Yaskawa INFORM job: A_ROOF_SIDE_0617_1_PL8.JBI

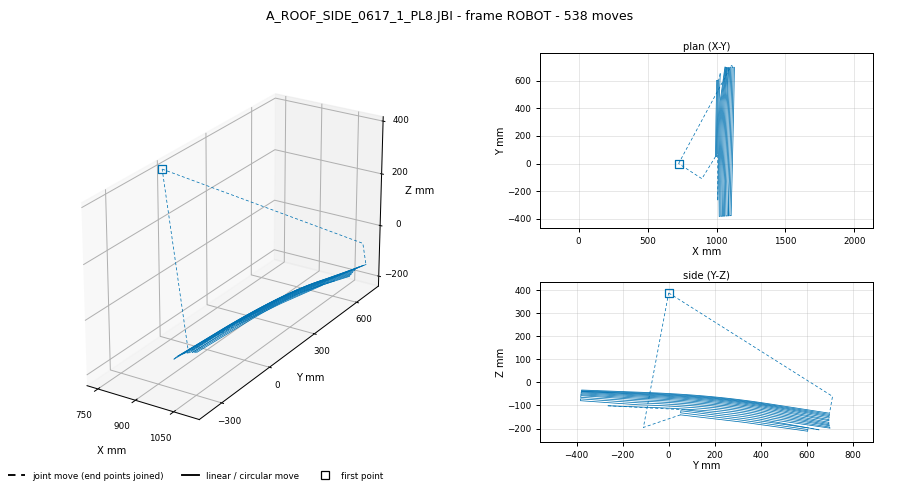
[picture p0: tool path of A_ROOF_SIDE_0617_1_PL8.JBI in frame ROBOT, 538 of 538 moves have a stored position in this frame; points joined in program order, loops and branches not executed]
/JOB
//NAME A_ROOF_SIDE_0617_1_PL8
//POS
///NPOS 538,0,0,0,0,0
///TOOL 0
///USER 0
///POSTYPE ROBOT
///RECTAN
///RCONF 1,0,0,0,0,0,0,0,0,0,0,0,0,0,0,0,0,0,0,0,0,0,0,0
C00000=725.000,0.000,388.500,-180.000,-0.000,0.000
///USER 0
///POSTYPE ROBOT
///RECTAN
C00001=1107.967,711.119,-60.351,170.013,-16.450,1.066
C00002=1129.814,698.090,-133.511,170.013,-16.450,1.066
C00003=1128.918,648.693,-125.824,170.280,-16.606,0.127
C00004=1125.127,440.216,-93.381,170.565,-16.222,-0.283
C00005=1124.690,417.893,-89.964,171.018,-15.554,-0.369
C00006=1124.432,405.287,-88.079,171.255,-15.284,-0.399
C00007=1124.145,391.687,-86.083,171.500,-15.059,-0.421
C00008=1123.832,377.143,-83.997,171.755,-14.880,-0.433
C00009=1123.494,361.710,-81.840,172.018,-14.745,-0.437
C00010=1123.153,346.326,-79.747,172.273,-14.658,-0.434
C00011=1122.809,330.942,-77.713,172.523,-14.609,-0.424
C00012=1122.428,313.994,-75.547,172.790,-14.590,-0.408
C00013=1122.033,296.572,-73.395,173.060,-14.603,-0.387
C00014=1121.637,279.197,-71.328,173.323,-14.640,-0.363
C00015=1121.232,261.424,-69.294,173.585,-14.699,-0.335
C00016=1120.814,243.073,-67.283,173.850,-14.777,-0.305
C00017=1120.393,224.685,-65.353,174.108,-14.866,-0.273
C00018=1119.732,195.801,-62.498,174.517,-15.066,-0.216
C00019=1119.265,175.675,-60.613,174.766,-15.231,-0.174
C00020=1118.801,155.633,-58.834,175.006,-15.376,-0.135
C00021=1118.319,134.585,-57.072,175.249,-15.506,-0.098
C00022=1117.837,113.529,-55.408,175.483,-15.610,-0.064
C00023=1117.332,91.368,-53.767,175.719,-15.694,-0.032
C00024=1116.829,69.300,-52.233,175.943,-15.752,-0.004
C00025=1116.302,46.128,-50.732,176.170,-15.788,0.023
C00026=1115.776,23.049,-49.338,176.385,-15.806,0.048
C00027=1115.222,-1.112,-47.980,176.600,-15.809,0.071
C00028=1114.667,-25.180,-46.725,176.803,-15.805,0.094
C00029=1114.080,-50.322,-45.510,177.003,-15.802,0.117
C00030=1113.487,-75.397,-44.389,177.192,-15.806,0.141
C00031=1112.880,-100.584,-43.344,177.368,-15.827,0.165
C00032=1107.242,-327.548,-34.722,177.586,-15.877,0.062
C00033=1106.000,-377.496,-32.825,177.740,-15.899,-0.498
C00034=1096.541,-377.841,-35.728,177.817,-15.909,-0.779
C00035=1097.765,-327.892,-37.635,177.577,-15.875,0.098
C00036=1103.334,-100.476,-46.316,177.367,-15.826,0.169
C00037=1103.941,-75.303,-47.364,177.191,-15.806,0.144
C00038=1104.536,-50.241,-48.492,177.002,-15.801,0.120
C00039=1105.124,-25.111,-49.715,176.802,-15.805,0.096
C00040=1105.682,-1.059,-50.978,176.599,-15.809,0.073
C00041=1106.238,23.090,-52.343,176.385,-15.805,0.049
C00042=1106.766,46.153,-53.742,176.170,-15.788,0.024
C00043=1107.294,69.311,-55.246,175.943,-15.752,-0.003
C00044=1107.796,91.366,-56.778,175.718,-15.694,-0.032
C00045=1108.299,113.513,-58.415,175.483,-15.610,-0.064
C00046=1108.778,134.556,-60.069,175.249,-15.506,-0.098
C00047=1109.257,155.591,-61.820,175.007,-15.376,-0.136
C00048=1109.716,175.621,-63.583,174.766,-15.231,-0.175
C00049=1110.177,195.736,-65.450,174.517,-15.066,-0.217
C00050=1110.476,208.693,-66.708,174.325,-14.951,-0.246
C00051=1110.835,224.601,-68.294,174.108,-14.866,-0.274
C00052=1111.254,242.975,-70.217,173.850,-14.777,-0.306
C00053=1111.671,261.313,-72.224,173.585,-14.700,-0.337
C00054=1112.076,279.073,-74.255,173.323,-14.641,-0.365
C00055=1112.471,296.435,-76.322,173.061,-14.603,-0.390
C00056=1112.868,313.842,-78.478,172.791,-14.591,-0.411
C00057=1113.252,330.775,-80.653,172.523,-14.609,-0.427
C00058=1113.600,346.143,-82.698,172.274,-14.659,-0.437
C00059=1113.947,361.511,-84.808,172.019,-14.746,-0.441
C00060=1114.293,376.928,-86.991,171.756,-14.880,-0.437
C00061=1114.616,391.453,-89.109,171.501,-15.060,-0.425
C00062=1114.916,405.034,-91.143,171.257,-15.285,-0.405
C00063=1115.190,417.620,-93.073,171.019,-15.554,-0.375
C00064=1115.441,429.264,-94.900,170.787,-15.869,-0.337
C00065=1115.665,439.899,-96.600,170.567,-16.223,-0.290
C00066=1119.956,648.127,-130.473,170.298,-16.616,0.066
C00067=1120.972,697.468,-138.499,169.874,-16.366,1.559
C00068=1112.130,696.831,-143.487,170.053,-16.473,0.925
C00069=1110.996,647.549,-135.122,170.327,-16.632,-0.034
C00070=1106.203,439.581,-99.820,170.569,-16.224,-0.297
C00071=1105.958,428.969,-98.061,170.789,-15.870,-0.343
C00072=1105.690,417.346,-96.183,171.021,-15.555,-0.381
C00073=1105.400,404.781,-94.207,171.258,-15.286,-0.410
C00074=1105.088,391.219,-92.134,171.502,-15.061,-0.430
C00075=1104.754,376.713,-89.984,171.758,-14.881,-0.441
C00076=1104.400,361.312,-87.777,172.020,-14.746,-0.445
C00077=1104.048,345.961,-85.648,172.275,-14.659,-0.440
C00078=1103.695,330.607,-83.592,172.524,-14.610,-0.430
C00079=1103.308,313.689,-81.408,172.791,-14.591,-0.413
C00080=1102.911,296.297,-79.249,173.061,-14.603,-0.392
C00081=1102.515,278.948,-77.182,173.324,-14.641,-0.367
C00082=1102.110,261.203,-75.154,173.586,-14.700,-0.339
C00083=1101.695,242.879,-73.151,173.850,-14.777,-0.308
C00084=1101.278,224.517,-71.234,174.109,-14.867,-0.275
C00085=1100.917,208.619,-69.643,174.325,-14.952,-0.247
C00086=1100.623,195.671,-68.402,174.517,-15.066,-0.218
C00087=1100.167,175.566,-66.553,174.767,-15.231,-0.175
C00088=1099.714,155.549,-64.805,175.007,-15.376,-0.136
C00089=1099.238,134.527,-63.067,175.249,-15.506,-0.098
C00090=1098.762,113.496,-61.421,175.483,-15.610,-0.064
C00091=1098.260,91.363,-59.788,175.718,-15.693,-0.031
C00092=1097.759,69.323,-58.260,175.943,-15.752,-0.002
C00093=1097.230,46.180,-56.752,176.169,-15.788,0.025
C00094=1096.700,23.129,-55.348,176.384,-15.805,0.050
C00095=1096.142,-1.005,-53.975,176.599,-15.809,0.075
C00096=1095.582,-25.044,-52.704,176.802,-15.805,0.098
C00097=1094.991,-50.159,-51.473,177.002,-15.801,0.123
C00098=1094.393,-75.207,-50.339,177.190,-15.806,0.148
C00099=1093.786,-100.367,-49.288,177.366,-15.826,0.173
C00100=1088.286,-328.237,-40.548,177.560,-15.873,0.157
C00101=1087.079,-378.186,-38.632,177.718,-15.896,-0.418
C00102=1088.610,-378.564,-38.329,177.695,-18.663,-0.346
C00103=1087.602,-328.640,-40.895,177.480,-18.637,0.327
C00104=1083.551,-128.437,-51.180,177.438,-18.638,0.450
C00105=1084.148,-103.852,-52.113,177.268,-18.642,0.435
C00106=1084.733,-79.664,-53.112,177.091,-18.674,0.423
C00107=1085.309,-55.600,-54.189,176.905,-18.731,0.414
C00108=1085.881,-31.455,-55.358,176.709,-18.808,0.406
C00109=1086.446,-7.402,-56.613,176.507,-18.895,0.400
C00110=1087.009,16.760,-57.969,176.295,-18.988,0.394
C00111=1087.541,39.825,-59.355,176.086,-19.073,0.389
C00112=1088.069,62.885,-60.834,175.869,-19.149,0.384
C00113=1088.598,86.051,-62.417,175.642,-19.211,0.377
C00114=1089.097,108.100,-64.017,175.419,-19.253,0.369
C00115=1089.596,130.256,-65.721,175.186,-19.276,0.358
C00116=1090.069,151.295,-67.432,174.954,-19.282,0.346
C00117=1090.541,172.325,-69.237,174.713,-19.270,0.332
C00118=1090.993,192.461,-71.058,174.472,-19.248,0.317
C00119=1091.350,208.411,-72.568,174.213,-19.225,0.305
C00120=1091.518,215.896,-73.306,174.110,-19.239,0.302
C00121=1091.934,234.336,-75.185,173.852,-19.278,0.297
C00122=1092.339,252.213,-77.095,173.593,-19.321,0.292
C00123=1092.756,270.561,-79.145,173.319,-19.373,0.289
C00124=1093.151,287.916,-81.174,173.051,-19.435,0.288
C00125=1093.539,304.875,-83.242,172.781,-19.511,0.289
C00126=1093.917,321.322,-85.330,172.510,-19.607,0.295
C00127=1094.297,337.735,-87.498,172.229,-19.729,0.304
C00128=1094.655,353.122,-89.610,171.955,-19.874,0.319
C00129=1094.993,367.519,-91.659,171.687,-20.045,0.338
C00130=1095.333,381.964,-93.787,171.405,-20.259,0.365
C00131=1095.657,395.520,-95.855,171.126,-20.509,0.400
C00132=1095.962,408.134,-97.843,170.850,-20.795,0.441
C00133=1096.246,419.755,-99.732,170.576,-21.115,0.490
C00134=1096.509,430.438,-101.522,170.302,-21.468,0.545
C00135=1096.760,440.397,-103.240,170.025,-21.859,0.609
C00136=1102.067,647.102,-139.894,169.706,-22.284,0.894
C00137=1103.328,696.318,-148.621,169.517,-22.199,1.393
C00138=1095.176,695.746,-154.761,168.937,-27.270,1.833
C00139=1093.722,646.605,-145.650,168.975,-27.285,1.750
C00140=1087.640,441.197,-107.568,169.355,-26.880,1.480
C00141=1087.362,431.351,-105.797,169.700,-26.465,1.400
C00142=1087.070,420.586,-103.925,170.040,-26.078,1.327
C00143=1086.786,409.872,-102.124,170.346,-25.748,1.265
C00144=1086.506,399.019,-100.357,170.629,-25.461,1.212
C00145=1086.184,386.323,-98.356,170.934,-25.175,1.160
C00146=1085.845,372.684,-96.281,171.239,-24.915,1.114
C00147=1085.515,359.148,-94.295,171.522,-24.696,1.075
C00148=1085.166,344.673,-92.247,171.808,-24.495,1.041
C00149=1084.806,329.574,-90.188,172.089,-24.315,1.010
C00150=1084.418,313.062,-88.024,172.381,-24.143,0.982
C00151=1084.033,296.553,-85.949,172.660,-23.990,0.958
C00152=1083.631,279.213,-83.859,172.941,-23.844,0.935
C00153=1083.216,261.139,-81.776,173.221,-23.701,0.914
C00154=1082.793,242.708,-79.747,173.496,-23.562,0.894
C00155=1082.371,224.240,-77.807,173.762,-23.423,0.875
C00156=1082.004,208.130,-76.188,173.986,-23.302,0.859
C00157=1081.621,191.051,-74.571,174.293,-23.234,0.850
C00158=1081.149,170.019,-72.671,174.543,-23.151,0.841
C00159=1080.675,148.977,-70.868,174.780,-23.062,0.831
C00160=1080.175,126.805,-69.067,175.017,-22.959,0.821
C00161=1079.674,104.750,-67.372,175.244,-22.845,0.809
C00162=1079.145,81.692,-65.701,175.472,-22.715,0.796
C00163=1078.611,58.504,-64.117,175.694,-22.574,0.783
C00164=1078.075,35.433,-62.636,175.908,-22.429,0.771
C00165=1077.532,12.237,-61.240,176.119,-22.282,0.759
C00166=1076.988,-10.831,-59.941,176.323,-22.141,0.748
C00167=1076.437,-33.998,-58.724,176.523,-22.011,0.740
C00168=1075.885,-57.066,-57.598,176.719,-21.901,0.734
C00169=1075.327,-80.143,-56.557,176.907,-21.815,0.731
C00170=1074.762,-103.356,-55.591,177.090,-21.760,0.731
C00171=1074.152,-128.448,-54.634,177.278,-21.736,0.736
C00172=1077.280,-329.161,-44.155,177.328,-21.727,0.620
C00173=1078.056,-379.088,-41.549,177.471,-21.743,0.235
C00174=1068.156,-379.602,-45.133,177.168,-25.215,0.859
C00175=1067.520,-329.679,-47.816,177.119,-25.210,0.975
C00176=1064.951,-128.477,-58.631,177.065,-25.228,1.072
C00177=1065.229,-116.921,-59.062,176.973,-25.231,1.075
C00178=1065.772,-94.813,-59.942,176.790,-25.259,1.081
C00179=1066.313,-72.653,-60.902,176.600,-25.321,1.092
C00180=1066.853,-50.507,-61.942,176.405,-25.414,1.106
C00181=1067.390,-28.375,-63.063,176.206,-25.532,1.124
C00182=1067.937,-5.743,-64.294,176.002,-25.673,1.145
C00183=1068.491,17.337,-65.640,175.791,-25.833,1.169
C00184=1069.042,40.486,-67.081,175.577,-26.003,1.196
C00185=1069.589,63.630,-68.614,175.359,-26.177,1.225
C00186=1070.132,86.767,-70.243,175.137,-26.351,1.254
C00187=1070.658,109.399,-71.931,174.912,-26.517,1.284
C00188=1071.167,131.459,-73.669,174.684,-26.676,1.314
C00189=1071.663,153.080,-75.466,174.451,-26.827,1.343
C00190=1072.145,174.194,-77.317,174.211,-26.973,1.373
C00191=1072.611,194.733,-79.211,173.962,-27.116,1.402
C00192=1072.907,207.781,-80.465,173.665,-27.213,1.423
C00193=1073.311,225.064,-82.231,173.424,-27.400,1.459
C00194=1073.745,243.621,-84.215,173.156,-27.596,1.499
C00195=1074.180,262.140,-86.287,172.876,-27.788,1.539
C00196=1074.609,280.284,-88.415,172.589,-27.977,1.580
C00197=1075.028,297.831,-90.565,172.298,-28.165,1.621
C00198=1075.427,314.433,-92.689,172.006,-28.354,1.663
C00199=1075.807,330.049,-94.772,171.717,-28.547,1.706
C00200=1076.185,345.347,-96.894,171.414,-28.755,1.752
C00201=1076.552,359.920,-98.998,171.105,-28.980,1.802
C00202=1076.903,373.558,-101.043,170.793,-29.218,1.856
C00203=1077.239,386.313,-103.027,170.477,-29.476,1.912
C00204=1077.533,397.166,-104.775,170.185,-29.725,1.968
C00205=1077.863,408.975,-106.743,169.837,-30.038,2.037
C00206=1078.176,419.800,-108.614,169.482,-30.369,2.110
C00207=1078.474,429.699,-110.386,169.121,-30.716,2.187
C00208=1078.782,439.524,-112.210,168.717,-31.114,2.275
C00209=1085.876,646.161,-151.960,168.189,-31.575,2.533
C00210=1087.559,695.233,-161.401,168.348,-31.628,2.229
C00211=1085.673,695.022,-166.146,167.623,-35.268,2.859
C00212=1082.684,645.978,-156.885,167.361,-35.185,3.314
C00213=1070.662,448.821,-119.660,167.510,-35.179,3.127
C00214=1070.296,439.181,-117.737,168.020,-34.766,3.021
C00215=1069.983,430.349,-116.040,168.434,-34.434,2.936
C00216=1069.647,420.308,-114.182,168.853,-34.101,2.851
C00217=1069.471,414.833,-113.197,169.061,-33.937,2.808
C00218=1069.131,403.873,-111.284,169.443,-33.640,2.731
C00219=1068.806,392.964,-109.447,169.785,-33.381,2.663
C00220=1068.464,381.099,-107.520,170.122,-33.133,2.597
C00221=1068.095,367.780,-105.438,170.467,-32.888,2.532
C00222=1067.724,354.051,-103.373,170.792,-32.666,2.471
C00223=1067.353,339.856,-101.319,171.102,-32.462,2.414
C00224=1066.964,324.712,-99.214,171.408,-32.264,2.358
C00225=1066.556,308.542,-97.054,171.711,-32.069,2.303
C00226=1066.142,291.850,-94.918,172.005,-31.880,2.250
C00227=1065.720,274.707,-92.814,172.288,-31.692,2.197
C00228=1065.281,256.709,-90.699,172.569,-31.496,2.143
C00229=1064.831,238.191,-88.620,172.845,-31.290,2.088
C00230=1064.475,223.486,-87.033,173.054,-31.121,2.045
C00231=1064.085,207.368,-85.358,173.275,-30.929,1.997
C00232=1063.829,196.371,-84.284,173.586,-30.836,1.971
C00233=1063.364,176.327,-82.401,173.836,-30.678,1.927
C00234=1062.893,156.134,-80.594,174.069,-30.525,1.884
C00235=1062.401,135.075,-78.801,174.300,-30.369,1.841
C00236=1061.880,113.012,-77.019,174.529,-30.207,1.797
C00237=1061.353,90.801,-75.318,174.751,-30.044,1.755
C00238=1060.799,67.727,-73.649,174.975,-29.877,1.712
C00239=1060.262,45.503,-72.130,175.186,-29.719,1.673
C00240=1059.725,23.413,-70.707,175.395,-29.569,1.635
C00241=1059.185,1.324,-69.370,175.602,-29.429,1.600
C00242=1058.639,-20.884,-68.111,175.812,-29.304,1.568
C00243=1058.095,-42.966,-66.946,176.018,-29.200,1.540
C00244=1057.574,-64.054,-65.913,176.216,-29.126,1.516
C00245=1057.052,-85.283,-64.950,176.412,-29.078,1.496
C00246=1056.555,-105.402,-64.111,176.594,-29.061,1.480
C00247=1055.993,-128.515,-63.229,176.797,-29.077,1.467
C00248=1058.090,-330.203,-52.056,176.852,-29.052,1.390
C00249=1058.608,-380.124,-49.292,176.773,-29.044,1.551
C00250=1050.380,-380.614,-53.513,176.302,-33.105,2.273
C00251=1049.775,-330.705,-56.474,176.539,-33.127,1.840
C00252=1047.327,-129.069,-68.445,176.478,-33.153,1.918
C00253=1047.362,-127.070,-68.526,176.459,-33.153,1.920
C00254=1047.879,-105.949,-69.326,176.261,-33.099,1.940
C00255=1048.393,-85.139,-70.194,176.061,-33.077,1.964
C00256=1048.903,-64.584,-71.130,175.861,-33.085,1.991
C00257=1049.429,-43.491,-72.170,175.654,-33.119,2.022
C00258=1049.956,-22.405,-73.293,175.448,-33.176,2.058
C00259=1050.512,-0.188,-74.563,175.233,-33.258,2.098
C00260=1051.064,21.906,-75.914,175.020,-33.355,2.141
C00261=1051.614,43.999,-77.354,174.810,-33.464,2.187
C00262=1052.164,66.232,-78.889,174.597,-33.581,2.235
C00263=1052.706,88.312,-80.504,174.383,-33.703,2.285
C00264=1053.247,110.530,-82.218,174.162,-33.830,2.336
C00265=1053.780,132.597,-84.016,173.934,-33.957,2.388
C00266=1054.285,153.658,-85.822,173.705,-34.082,2.440
C00267=1054.763,173.716,-87.630,173.473,-34.206,2.491
C00268=1055.225,193.096,-89.463,173.230,-34.334,2.542
C00269=1055.554,206.894,-90.825,172.843,-34.435,2.581
C00270=1055.703,212.785,-91.440,172.766,-34.500,2.602
C00271=1056.202,232.613,-93.575,172.496,-34.711,2.671
C00272=1056.671,251.300,-95.681,172.227,-34.899,2.736
C00273=1057.120,269.057,-97.770,171.956,-35.072,2.797
C00274=1057.572,286.820,-99.954,171.667,-35.245,2.860
C00275=1058.004,303.622,-102.108,171.375,-35.412,2.921
C00276=1058.420,319.514,-104.233,171.076,-35.578,2.982
C00277=1058.816,334.373,-106.302,170.775,-35.745,3.042
C00278=1059.221,349.205,-108.450,170.448,-35.929,3.106
C00279=1059.611,363.053,-110.539,170.112,-36.121,3.172
C00280=1059.987,375.974,-112.567,169.769,-36.324,3.238
C00281=1060.351,388.020,-114.531,169.415,-36.538,3.307
C00282=1060.725,399.843,-116.535,169.029,-36.777,3.382
C00283=1061.093,410.950,-118.492,168.625,-37.034,3.461
C00284=1061.448,421.083,-120.350,168.210,-37.301,3.541
C00285=1061.790,430.304,-122.105,167.786,-37.574,3.622
C00286=1062.137,439.125,-123.850,167.329,-37.867,3.709
C00287=1062.510,447.936,-125.662,166.813,-38.196,3.805
C00288=1075.955,645.876,-163.643,166.601,-38.231,3.971
C00289=1079.282,694.871,-173.044,167.101,-38.379,3.164
C00290=1075.415,695.159,-178.337,166.551,-40.986,3.567
C00291=1071.311,646.171,-169.207,165.871,-40.794,4.606
C00292=1054.724,448.260,-132.325,166.101,-40.779,4.434
C00293=1054.610,446.311,-131.924,166.230,-40.722,4.414
C00294=1054.216,437.743,-130.128,166.759,-40.461,4.326
C00295=1053.840,428.947,-128.357,167.239,-40.220,4.244
C00296=1053.448,419.135,-126.460,167.713,-39.981,4.161
C00297=1053.061,408.824,-124.545,168.154,-39.759,4.081
C00298=1052.661,397.544,-122.535,168.582,-39.546,4.003
C00299=1052.286,386.328,-120.613,168.963,-39.360,3.932
C00300=1051.899,374.242,-118.621,169.332,-39.185,3.863
C00301=1051.506,361.410,-116.588,169.686,-39.023,3.795
C00302=1051.093,347.398,-114.456,170.034,-38.867,3.728
C00303=1050.695,333.396,-112.407,170.350,-38.730,3.665
C00304=1050.274,318.188,-110.271,170.663,-38.597,3.601
C00305=1049.840,302.168,-108.112,170.966,-38.470,3.537
C00306=1049.388,285.212,-105.920,171.260,-38.344,3.472
C00307=1048.917,267.295,-103.701,171.545,-38.216,3.406
C00308=1048.448,249.385,-101.576,171.812,-38.088,3.341
C00309=1047.955,230.394,-99.417,172.076,-37.947,3.271
C00310=1047.327,206.362,-96.817,172.388,-37.756,3.183
C00311=1046.886,188.254,-95.024,172.868,-37.679,3.129
C00312=1046.398,168.205,-93.133,173.114,-37.609,3.074
C00313=1045.906,147.976,-91.318,173.343,-37.549,3.021
C00314=1045.370,126.086,-89.451,173.574,-37.490,2.965
C00315=1044.822,103.869,-87.653,173.797,-37.436,2.909
C00316=1044.273,81.793,-85.961,174.011,-37.389,2.856
C00317=1043.717,59.563,-84.348,174.222,-37.345,2.803
C00318=1043.160,37.472,-82.836,174.431,-37.309,2.753
C00319=1042.600,15.376,-81.412,174.641,-37.283,2.704
C00320=1042.062,-5.859,-80.127,174.847,-37.271,2.660
C00321=1041.529,-26.948,-78.935,175.054,-37.274,2.618
C00322=1040.998,-48.038,-77.827,175.265,-37.297,2.579
C00323=1040.491,-68.268,-76.845,175.469,-37.340,2.546
C00324=1040.009,-87.770,-75.972,175.666,-37.403,2.516
C00325=1039.525,-107.511,-75.164,175.862,-37.492,2.490
C00326=1039.019,-128.637,-74.379,176.069,-37.612,2.465
C00327=1039.019,-130.639,-74.273,176.091,-37.597,2.459
C00328=1042.796,-331.146,-60.722,176.172,-37.585,2.342
C00329=1043.735,-381.023,-57.351,175.752,-37.547,3.030
C00330=1034.148,-381.660,-64.410,174.884,-42.656,4.164
C00331=1033.551,-331.772,-67.694,175.679,-42.727,2.993
C00332=1031.136,-130.219,-80.966,175.534,-42.747,3.179
C00333=1031.153,-128.221,-81.060,175.512,-42.747,3.184
C00334=1031.650,-107.095,-81.818,175.304,-42.533,3.211
C00335=1032.134,-86.912,-82.625,175.103,-42.349,3.240
C00336=1032.601,-67.720,-83.470,174.909,-42.193,3.270
C00337=1033.099,-47.622,-84.433,174.709,-42.047,3.304
C00338=1033.627,-26.531,-85.530,174.501,-41.912,3.342
C00339=1034.159,-5.442,-86.714,174.299,-41.793,3.382
C00340=1034.696,15.792,-87.993,174.100,-41.685,3.423
C00341=1035.256,37.888,-89.413,173.898,-41.585,3.468
C00342=1035.815,59.979,-90.923,173.700,-41.493,3.514
C00343=1036.374,82.208,-92.534,173.500,-41.408,3.561
C00344=1036.925,104.283,-94.226,173.298,-41.329,3.608
C00345=1037.475,126.498,-96.025,173.086,-41.255,3.656
C00346=1037.994,147.563,-97.823,172.874,-41.191,3.702
C00347=1038.485,167.621,-99.624,172.657,-41.138,3.748
C00348=1038.952,186.675,-101.420,172.431,-41.098,3.792
C00349=1039.422,205.776,-103.312,171.906,-41.073,3.840
C00350=1039.748,217.949,-104.621,171.762,-41.107,3.881
C00351=1040.266,237.334,-106.782,171.517,-41.157,3.946
C00352=1040.776,256.419,-109.002,171.256,-41.205,4.009
C00353=1041.261,274.492,-111.199,170.989,-41.253,4.070
C00354=1041.732,291.856,-113.401,170.707,-41.305,4.131
C00355=1042.178,308.054,-115.544,170.419,-41.362,4.190
C00356=1042.606,323.271,-117.642,170.122,-41.428,4.248
C00357=1043.016,337.469,-119.679,169.817,-41.501,4.305
C00358=1043.439,351.642,-121.796,169.481,-41.590,4.367
C00359=1043.848,364.836,-123.849,169.134,-41.691,4.429
C00360=1044.253,377.292,-125.865,168.770,-41.804,4.493
C00361=1044.650,388.936,-127.825,168.390,-41.929,4.558
C00362=1045.060,400.331,-129.823,167.976,-42.072,4.627
C00363=1045.460,410.809,-131.736,167.549,-42.225,4.697
C00364=1045.848,420.326,-133.543,167.115,-42.384,4.766
C00365=1046.229,429.149,-135.284,166.663,-42.550,4.836
C00366=1046.627,437.750,-137.049,166.170,-42.730,4.910
C00367=1047.072,446.538,-138.922,165.600,-42.934,4.991
C00368=1047.249,448.876,-139.385,165.439,-42.977,5.010
C00369=1066.928,646.790,-174.714,165.187,-42.971,5.194
C00370=1071.798,695.777,-183.459,166.051,-43.207,3.929
C00371=1069.075,696.775,-187.811,165.209,-45.018,4.817
C00372=1063.320,647.778,-179.671,164.552,-44.840,5.748
C00373=1040.136,450.401,-146.879,164.791,-44.875,5.544
C00374=1039.899,448.024,-146.449,164.960,-44.859,5.532
C00375=1039.744,446.069,-146.061,165.098,-44.838,5.519
C00376=1039.469,441.195,-145.009,165.429,-44.764,5.482
C00377=1039.049,432.917,-143.258,165.942,-44.644,5.419
C00378=1038.624,423.939,-141.435,166.439,-44.530,5.357
C00379=1038.206,414.429,-139.582,166.906,-44.425,5.296
C00380=1037.793,404.418,-137.707,167.344,-44.331,5.236
C00381=1037.372,393.517,-135.748,167.770,-44.246,5.176
C00382=1036.954,381.992,-133.759,168.172,-44.177,5.119
C00383=1036.553,370.344,-131.829,168.536,-44.124,5.066
C00384=1036.140,357.737,-129.821,168.890,-44.085,5.014
C00385=1035.723,344.362,-127.775,169.226,-44.062,4.963
C00386=1035.307,330.485,-125.736,169.540,-44.056,4.915
C00387=1034.875,315.583,-123.634,169.843,-44.065,4.867
C00388=1034.441,300.182,-121.550,170.126,-44.092,4.822
C00389=1033.997,284.121,-119.464,170.392,-44.133,4.778
C00390=1033.535,267.126,-117.347,170.647,-44.192,4.734
C00391=1033.302,258.494,-116.305,170.767,-44.226,4.713
C00392=1032.811,240.223,-114.169,171.003,-44.307,4.670
C00393=1032.320,221.918,-112.117,171.219,-44.399,4.628
C00394=1031.868,205.136,-110.309,171.400,-44.491,4.591
C00395=1031.660,196.583,-109.458,171.817,-44.573,4.581
C00396=1031.223,178.502,-107.722,172.024,-44.760,4.560
C00397=1030.766,159.446,-105.980,172.220,-44.967,4.540
C00398=1030.284,139.384,-104.235,172.407,-45.195,4.518
C00399=1030.031,128.853,-103.354,172.499,-45.316,4.507
C00400=1029.493,106.642,-101.572,172.684,-45.578,4.483
C00401=1028.954,84.568,-99.897,172.860,-45.841,4.458
C00402=1028.412,62.487,-98.315,173.032,-46.108,4.432
C00403=1027.862,40.254,-96.815,173.206,-46.380,4.404
C00404=1027.316,18.160,-95.415,173.383,-46.655,4.375
C00405=1026.771,-3.934,-94.109,173.567,-46.935,4.346
C00406=1026.250,-25.153,-92.944,173.751,-47.213,4.318
C00407=1025.739,-46.241,-91.875,173.940,-47.498,4.290
///RCONF 1,0,0,1,0,0,0,0,0,0,0,0,0,0,0,0,0,0,0,0,0,0,0,0
C00408=1025.258,-66.336,-90.941,174.125,-47.779,4.264
///RCONF 1,0,0,1,1,0,0,0,0,0,0,0,0,0,0,0,0,0,0,0,0,0,0,0
C00409=1024.786,-86.462,-90.086,174.313,-48.071,4.238
///RCONF 1,0,0,0,1,0,0,0,0,0,0,0,0,0,0,0,0,0,0,0,0,0,0,0
C00410=1024.323,-106.699,-89.312,174.503,-48.376,4.214
C00411=1023.834,-128.823,-88.559,174.709,-48.720,4.188
C00412=1023.821,-130.821,-88.459,174.731,-48.722,4.180
C00413=1025.992,-332.340,-74.658,175.012,-48.713,3.829
C00414=1026.529,-382.220,-71.243,174.452,-48.667,4.575
C00415=1019.498,-382.803,-79.194,173.561,-55.852,5.565
C00416=1019.052,-332.929,-82.718,173.951,-55.881,5.094
C00417=1017.248,-131.438,-96.963,173.391,-55.871,5.752
C00418=1017.257,-129.440,-97.066,173.367,-55.866,5.763
C00419=1017.738,-105.325,-97.824,173.192,-55.315,5.766
C00420=1018.183,-84.083,-98.580,173.039,-54.821,5.765
///RCONF 1,0,0,0,0,0,0,0,0,0,0,0,0,0,0,0,0,0,0,0,0,0,0,0
C00421=1018.638,-62.987,-99.424,172.889,-54.332,5.763
///RCONF 1,0,0,1,0,0,0,0,0,0,0,0,0,0,0,0,0,0,0,0,0,0,0,0
C00422=1019.104,-41.900,-100.358,172.745,-53.845,5.758
C00423=1019.583,-20.701,-101.388,172.607,-53.357,5.752
C00424=1020.087,1.387,-102.556,172.473,-52.845,5.741
///RCONF 1,0,0,0,0,0,0,0,0,0,0,0,0,0,0,0,0,0,0,0,0,0,0,0
C00425=1020.595,23.477,-103.819,172.349,-52.328,5.726
C00426=1021.085,44.706,-105.121,172.236,-51.829,5.709
C00427=1021.593,66.792,-106.564,172.123,-51.307,5.686
C00428=1022.106,89.187,-108.124,172.009,-50.776,5.660
C00429=1022.580,110.082,-109.668,171.899,-50.282,5.633
C00430=1023.054,131.150,-111.314,171.779,-49.787,5.604
C00431=1023.291,141.680,-112.171,171.713,-49.540,5.588
C00432=1023.741,161.741,-113.871,171.575,-49.075,5.558
C00433=1024.159,180.367,-115.535,171.427,-48.650,5.529
C00434=1024.534,196.944,-117.091,171.274,-48.280,5.504
C00435=1024.706,204.427,-117.817,170.851,-48.118,5.494
C00436=1024.904,212.022,-118.612,170.785,-47.987,5.492
C00437=1025.361,229.566,-120.504,170.618,-47.702,5.490
C00438=1025.792,246.077,-122.360,170.441,-47.457,5.494
C00439=1026.224,262.556,-124.286,170.243,-47.236,5.502
C00440=1026.652,278.632,-126.245,170.026,-47.039,5.514
C00441=1027.044,293.168,-128.089,169.807,-46.881,5.529
C00442=1027.447,307.766,-130.013,169.562,-46.741,5.548
C00443=1027.862,322.374,-132.019,169.289,-46.619,5.572
C00444=1028.239,335.238,-133.857,169.020,-46.529,5.597
C00445=1028.638,348.296,-135.796,168.717,-46.454,5.627
C00446=1029.057,361.389,-137.821,168.379,-46.397,5.661
C00447=1029.480,373.972,-139.851,168.013,-46.360,5.698
C00448=1029.898,385.641,-141.813,167.633,-46.343,5.738
C00449=1030.308,396.456,-143.707,167.240,-46.342,5.778
C00450=1030.747,407.267,-145.679,166.799,-46.357,5.823
C00451=1031.178,417.159,-147.562,166.346,-46.385,5.868
C00452=1031.643,427.078,-149.532,165.833,-46.426,5.917
C00453=1032.088,435.882,-151.358,165.321,-46.474,5.965
C00454=1032.587,444.804,-153.280,164.735,-46.531,6.015
C00455=1032.816,447.658,-153.848,164.535,-46.537,6.027
C00456=1033.123,450.597,-154.371,164.323,-46.530,6.036
C00457=1058.402,649.116,-185.768,163.979,-46.471,6.258
C00458=1064.641,698.116,-193.519,164.426,-46.591,5.642
C00459=1061.191,699.863,-198.268,163.777,-47.998,6.326
C00460=1054.326,650.852,-191.146,163.461,-47.914,6.752
C00461=1026.453,451.856,-162.234,163.870,-48.016,6.506
C00462=1026.106,448.912,-161.750,164.084,-48.058,6.509
C00463=1025.824,445.974,-161.209,164.290,-48.088,6.507
C00464=1025.607,443.047,-160.613,164.491,-48.105,6.501
C00465=1025.131,434.541,-158.786,165.034,-48.131,6.476
C00466=1024.663,425.396,-156.902,165.553,-48.165,6.450
C00467=1024.199,415.593,-154.970,166.046,-48.210,6.424
C00468=1023.756,405.449,-153.055,166.500,-48.266,6.400
C00469=1023.349,395.451,-151.244,166.900,-48.335,6.381
C00470=1022.937,384.623,-149.361,167.287,-48.422,6.362
C00471=1022.515,372.743,-147.380,167.665,-48.534,6.347
C00472=1022.120,360.938,-145.493,168.000,-48.663,6.336
C00473=1021.718,348.162,-143.535,168.322,-48.821,6.330
C00474=1021.336,335.363,-141.653,168.608,-49.001,6.329
C00475=1020.996,323.485,-139.972,168.846,-49.186,6.333
C00476=1020.617,309.660,-138.091,169.095,-49.423,6.343
C00477=1020.251,295.850,-136.288,169.313,-49.685,6.359
C00478=1019.873,281.108,-134.440,169.518,-49.992,6.384
C00479=1019.505,266.407,-132.672,169.696,-50.327,6.417
C00480=1019.144,251.716,-130.976,169.850,-50.694,6.457
C00481=1018.765,236.016,-129.237,169.989,-51.120,6.510
C00482=1018.414,221.279,-127.668,170.099,-51.556,6.569
C00483=1017.996,203.650,-125.873,170.203,-52.126,6.654
C00484=1017.848,196.178,-125.184,170.628,-52.407,6.702
C00485=1017.527,179.614,-123.711,170.698,-53.051,6.815
C00486=1017.179,161.491,-122.181,170.746,-53.762,6.940
C00487=1016.815,142.426,-120.657,170.772,-54.520,7.075
C00488=1016.433,122.358,-119.140,170.777,-55.320,7.217
C00489=1016.048,102.285,-117.707,170.767,-56.122,7.359
C00490=1015.640,81.146,-116.286,170.744,-56.962,7.508
C00491=1015.209,59.005,-114.891,170.714,-57.831,7.660
C00492=1014.777,36.860,-113.589,170.687,-58.676,7.804
C00493=1014.334,14.212,-112.354,170.670,-59.505,7.938
C00494=1013.894,-8.370,-111.217,170.672,-60.278,8.052
C00495=1013.468,-30.497,-110.199,170.702,-60.969,8.136
///RCONF 1,0,0,1,0,0,0,0,0,0,0,0,0,0,0,0,0,0,0,0,0,0,0,0
C00496=1013.049,-52.510,-109.278,170.769,-61.570,8.184
///RCONF 1,0,0,0,1,0,0,0,0,0,0,0,0,0,0,0,0,0,0,0,0,0,0,0
C00497=1009.105,-263.254,-101.142,172.129,-61.938,6.703
///RCONF 1,0,0,0,0,0,0,0,0,0,0,0,0,0,0,0,0,0,0,0,0,0,0,0
C00498=1008.805,68.226,-118.358,169.998,-53.543,6.326
C00499=1013.251,273.640,-141.883,169.067,-53.415,7.485
C00500=1013.562,287.560,-143.530,168.923,-52.940,7.395
C00501=1013.863,300.529,-145.130,168.763,-52.526,7.321
C00502=1014.180,313.561,-146.806,168.576,-52.139,7.255
C00503=1014.513,326.608,-148.557,168.359,-51.778,7.199
C00504=1014.865,339.629,-150.382,168.111,-51.444,7.150
C00505=1015.204,351.500,-152.116,167.853,-51.162,7.112
C00506=1015.571,363.500,-153.945,167.559,-50.896,7.080
C00507=1015.930,374.531,-155.697,167.254,-50.669,7.056
C00508=1016.317,385.642,-157.535,166.909,-50.457,7.035
C00509=1016.724,396.472,-159.407,166.531,-50.264,7.020
C00510=1025.080,603.016,-196.616,165.673,-50.001,7.623
C00511=1027.068,652.184,-205.476,165.727,-50.013,7.553
C00512=1015.679,604.810,-197.288,166.753,-52.476,8.643
C00513=1014.350,555.348,-190.098,166.832,-52.490,8.544
C00514=1008.694,344.979,-159.525,167.820,-52.945,7.715
C00515=1008.389,332.730,-157.823,168.067,-53.287,7.775
C00516=1008.234,326.097,-156.932,168.189,-53.479,7.810
C00517=1007.938,312.830,-155.213,168.409,-53.876,7.883
C00518=1003.565,102.555,-129.139,169.525,-54.376,6.791
C00519=1002.532,52.946,-122.989,169.762,-54.407,6.499
C00520=997.705,51.941,-131.798,169.760,-54.407,6.502
C00521=998.522,101.574,-137.792,169.524,-54.376,6.792
C00522=1001.985,311.911,-163.195,168.416,-53.877,7.875
C00523=1002.222,325.146,-164.867,168.196,-53.480,7.801
C00524=1002.347,331.784,-165.735,168.075,-53.288,7.766
C00525=1002.604,344.003,-167.396,167.828,-52.946,7.705
C00526=1007.490,554.438,-197.377,166.856,-52.494,8.514
C00527=1008.639,603.925,-204.429,166.777,-52.480,8.613
C00528=1001.592,603.037,-211.566,166.800,-52.485,8.583
C00529=1000.625,553.526,-204.653,166.879,-52.499,8.485
C00530=996.514,343.026,-175.268,167.837,-52.947,7.695
C00531=996.305,330.838,-173.646,168.083,-53.289,7.756
C00532=996.212,324.197,-172.803,168.203,-53.482,7.792
C00533=996.031,310.992,-171.177,168.423,-53.878,7.867
C00534=993.485,100.597,-146.449,169.523,-54.376,6.793
C00535=992.884,50.942,-140.613,169.757,-54.406,6.505
///RCONF 1,0,0,1,0,0,0,0,0,0,0,0,0,0,0,0,0,0,0,0,0,0,0,0
C00536=893.946,-109.711,-195.206,170.290,-54.473,5.850
///USER 0
///POSTYPE ROBOT
///RECTAN
///RCONF 1,0,0,0,0,0,0,0,0,0,0,0,0,0,0,0,0,0,0,0,0,0,0,0
C00537=725.000,0.000,388.500,-180.000,-0.000,0.000
//INST
///DATE 2021/06/17 09:36
///ATTR SC,RW,RJ
////FRAME ROBOT
///GROUP1 RB1
NOP
MOVJ C00000 VJ=100.00 PL=0
'Path Start: Op_ID_1
MOVJ C00001 VJ=25.00 PL=0
MOVJ C00002 VJ=25.00 PL=0
MOVL C00003 V=800.0 PL=8
SPYON
MOVL C00004 V=800.0 PL=8
MOVL C00005 V=800.0 PL=8
MOVL C00006 V=800.0 PL=8
MOVL C00007 V=800.0 PL=8
MOVL C00008 V=800.0 PL=8
MOVL C00009 V=800.0 PL=8
MOVL C00010 V=800.0 PL=8
MOVL C00011 V=800.0 PL=8
MOVL C00012 V=800.0 PL=8
MOVL C00013 V=800.0 PL=8
MOVL C00014 V=800.0 PL=8
MOVL C00015 V=800.0 PL=8
MOVL C00016 V=800.0 PL=8
MOVL C00017 V=800.0 PL=8
MOVL C00018 V=800.0 PL=8
MOVL C00019 V=800.0 PL=8
MOVL C00020 V=800.0 PL=8
MOVL C00021 V=800.0 PL=8
MOVL C00022 V=800.0 PL=8
MOVL C00023 V=800.0 PL=8
MOVL C00024 V=800.0 PL=8
MOVL C00025 V=800.0 PL=8
MOVL C00026 V=800.0 PL=8
MOVL C00027 V=800.0 PL=8
MOVL C00028 V=800.0 PL=8
MOVL C00029 V=800.0 PL=8
MOVL C00030 V=800.0 PL=8
MOVL C00031 V=800.0 PL=8
MOVL C00032 V=800.0 PL=8
SPYOF
MOVL C00033 V=800.0 PL=0
MOVJ C00034 VJ=25.00 PL=0
MOVL C00035 V=800.0 PL=8
SPYON
MOVL C00036 V=800.0 PL=8
MOVL C00037 V=800.0 PL=8
MOVL C00038 V=800.0 PL=8
MOVL C00039 V=800.0 PL=8
MOVL C00040 V=800.0 PL=8
MOVL C00041 V=800.0 PL=8
MOVL C00042 V=800.0 PL=8
MOVL C00043 V=800.0 PL=8
MOVL C00044 V=800.0 PL=8
MOVL C00045 V=800.0 PL=8
MOVL C00046 V=800.0 PL=8
MOVL C00047 V=800.0 PL=8
MOVL C00048 V=800.0 PL=8
MOVL C00049 V=800.0 PL=8
MOVL C00050 V=800.0 PL=8
MOVL C00051 V=800.0 PL=8
MOVL C00052 V=800.0 PL=8
MOVL C00053 V=800.0 PL=8
MOVL C00054 V=800.0 PL=8
MOVL C00055 V=800.0 PL=8
MOVL C00056 V=800.0 PL=8
MOVL C00057 V=800.0 PL=8
MOVL C00058 V=800.0 PL=8
MOVL C00059 V=800.0 PL=8
MOVL C00060 V=800.0 PL=8
MOVL C00061 V=800.0 PL=8
MOVL C00062 V=800.0 PL=8
MOVL C00063 V=800.0 PL=8
MOVL C00064 V=800.0 PL=8
MOVL C00065 V=800.0 PL=8
MOVL C00066 V=800.0 PL=8
SPYOF
MOVL C00067 V=800.0 PL=0
MOVJ C00068 VJ=25.00 PL=0
MOVL C00069 V=800.0 PL=8
SPYON
MOVL C00070 V=800.0 PL=8
MOVL C00071 V=800.0 PL=8
MOVL C00072 V=800.0 PL=8
MOVL C00073 V=800.0 PL=8
MOVL C00074 V=800.0 PL=8
MOVL C00075 V=800.0 PL=8
MOVL C00076 V=800.0 PL=8
MOVL C00077 V=800.0 PL=8
MOVL C00078 V=800.0 PL=8
MOVL C00079 V=800.0 PL=8
MOVL C00080 V=800.0 PL=8
MOVL C00081 V=800.0 PL=8
MOVL C00082 V=800.0 PL=8
MOVL C00083 V=800.0 PL=8
MOVL C00084 V=800.0 PL=8
MOVL C00085 V=800.0 PL=8
MOVL C00086 V=800.0 PL=8
MOVL C00087 V=800.0 PL=8
MOVL C00088 V=800.0 PL=8
MOVL C00089 V=800.0 PL=8
MOVL C00090 V=800.0 PL=8
MOVL C00091 V=800.0 PL=8
MOVL C00092 V=800.0 PL=8
MOVL C00093 V=800.0 PL=8
MOVL C00094 V=800.0 PL=8
MOVL C00095 V=800.0 PL=8
MOVL C00096 V=800.0 PL=8
MOVL C00097 V=800.0 PL=8
MOVL C00098 V=800.0 PL=8
MOVL C00099 V=800.0 PL=8
MOVL C00100 V=800.0 PL=8
SPYOF
MOVL C00101 V=800.0 PL=0
MOVJ C00102 VJ=25.00 PL=0
MOVL C00103 V=800.0 PL=8
SPYON
MOVL C00104 V=800.0 PL=8
MOVL C00105 V=800.0 PL=8
MOVL C00106 V=800.0 PL=8
MOVL C00107 V=800.0 PL=8
MOVL C00108 V=800.0 PL=8
MOVL C00109 V=800.0 PL=8
MOVL C00110 V=800.0 PL=8
MOVL C00111 V=800.0 PL=8
MOVL C00112 V=800.0 PL=8
MOVL C00113 V=800.0 PL=8
MOVL C00114 V=800.0 PL=8
MOVL C00115 V=800.0 PL=8
MOVL C00116 V=800.0 PL=8
MOVL C00117 V=800.0 PL=8
MOVL C00118 V=800.0 PL=8
MOVL C00119 V=800.0 PL=8
MOVL C00120 V=800.0 PL=8
MOVL C00121 V=800.0 PL=8
MOVL C00122 V=800.0 PL=8
MOVL C00123 V=800.0 PL=8
MOVL C00124 V=800.0 PL=8
MOVL C00125 V=800.0 PL=8
MOVL C00126 V=800.0 PL=8
MOVL C00127 V=800.0 PL=8
MOVL C00128 V=800.0 PL=8
MOVL C00129 V=800.0 PL=8
MOVL C00130 V=800.0 PL=8
MOVL C00131 V=800.0 PL=8
MOVL C00132 V=800.0 PL=8
MOVL C00133 V=800.0 PL=8
MOVL C00134 V=800.0 PL=8
MOVL C00135 V=800.0 PL=8
MOVL C00136 V=800.0 PL=8
SPYOF
MOVL C00137 V=800.0 PL=0
MOVJ C00138 VJ=25.00 PL=0
MOVL C00139 V=800.0 PL=8
SPYON
MOVL C00140 V=800.0 PL=8
MOVL C00141 V=800.0 PL=8
MOVL C00142 V=800.0 PL=8
MOVL C00143 V=800.0 PL=8
MOVL C00144 V=800.0 PL=8
MOVL C00145 V=800.0 PL=8
MOVL C00146 V=800.0 PL=8
MOVL C00147 V=800.0 PL=8
MOVL C00148 V=800.0 PL=8
MOVL C00149 V=800.0 PL=8
MOVL C00150 V=800.0 PL=8
MOVL C00151 V=800.0 PL=8
MOVL C00152 V=800.0 PL=8
MOVL C00153 V=800.0 PL=8
MOVL C00154 V=800.0 PL=8
MOVL C00155 V=800.0 PL=8
MOVL C00156 V=800.0 PL=8
MOVL C00157 V=800.0 PL=8
MOVL C00158 V=800.0 PL=8
MOVL C00159 V=800.0 PL=8
MOVL C00160 V=800.0 PL=8
MOVL C00161 V=800.0 PL=8
MOVL C00162 V=800.0 PL=8
MOVL C00163 V=800.0 PL=8
MOVL C00164 V=800.0 PL=8
MOVL C00165 V=800.0 PL=8
MOVL C00166 V=800.0 PL=8
MOVL C00167 V=800.0 PL=8
MOVL C00168 V=800.0 PL=8
MOVL C00169 V=800.0 PL=8
MOVL C00170 V=800.0 PL=8
MOVL C00171 V=800.0 PL=8
MOVL C00172 V=800.0 PL=8
SPYOF
MOVL C00173 V=800.0 PL=0
MOVJ C00174 VJ=25.00 PL=0
MOVL C00175 V=800.0 PL=8
SPYON
MOVL C00176 V=800.0 PL=8
MOVL C00177 V=800.0 PL=8
MOVL C00178 V=800.0 PL=8
MOVL C00179 V=800.0 PL=8
MOVL C00180 V=800.0 PL=8
MOVL C00181 V=800.0 PL=8
MOVL C00182 V=800.0 PL=8
MOVL C00183 V=800.0 PL=8
MOVL C00184 V=800.0 PL=8
MOVL C00185 V=800.0 PL=8
MOVL C00186 V=800.0 PL=8
MOVL C00187 V=800.0 PL=8
MOVL C00188 V=800.0 PL=8
MOVL C00189 V=800.0 PL=8
MOVL C00190 V=800.0 PL=8
MOVL C00191 V=800.0 PL=8
MOVL C00192 V=800.0 PL=8
MOVL C00193 V=800.0 PL=8
MOVL C00194 V=800.0 PL=8
MOVL C00195 V=800.0 PL=8
MOVL C00196 V=800.0 PL=8
MOVL C00197 V=800.0 PL=8
MOVL C00198 V=800.0 PL=8
MOVL C00199 V=800.0 PL=8
MOVL C00200 V=800.0 PL=8
MOVL C00201 V=800.0 PL=8
MOVL C00202 V=800.0 PL=8
MOVL C00203 V=800.0 PL=8
MOVL C00204 V=800.0 PL=8
MOVL C00205 V=800.0 PL=8
MOVL C00206 V=800.0 PL=8
MOVL C00207 V=800.0 PL=8
MOVL C00208 V=800.0 PL=8
MOVL C00209 V=800.0 PL=8
SPYOF
MOVL C00210 V=800.0 PL=0
MOVJ C00211 VJ=25.00 PL=0
MOVL C00212 V=800.0 PL=8
SPYON
MOVL C00213 V=800.0 PL=8
MOVL C00214 V=800.0 PL=8
MOVL C00215 V=800.0 PL=8
MOVL C00216 V=800.0 PL=8
MOVL C00217 V=800.0 PL=8
MOVL C00218 V=800.0 PL=8
MOVL C00219 V=800.0 PL=8
MOVL C00220 V=800.0 PL=8
MOVL C00221 V=800.0 PL=8
MOVL C00222 V=800.0 PL=8
MOVL C00223 V=800.0 PL=8
MOVL C00224 V=800.0 PL=8
MOVL C00225 V=800.0 PL=8
MOVL C00226 V=800.0 PL=8
MOVL C00227 V=800.0 PL=8
MOVL C00228 V=800.0 PL=8
MOVL C00229 V=800.0 PL=8
MOVL C00230 V=800.0 PL=8
MOVL C00231 V=800.0 PL=8
MOVL C00232 V=800.0 PL=8
MOVL C00233 V=800.0 PL=8
MOVL C00234 V=800.0 PL=8
MOVL C00235 V=800.0 PL=8
MOVL C00236 V=800.0 PL=8
MOVL C00237 V=800.0 PL=8
MOVL C00238 V=800.0 PL=8
MOVL C00239 V=800.0 PL=8
MOVL C00240 V=800.0 PL=8
MOVL C00241 V=800.0 PL=8
MOVL C00242 V=800.0 PL=8
MOVL C00243 V=800.0 PL=8
MOVL C00244 V=800.0 PL=8
MOVL C00245 V=800.0 PL=8
MOVL C00246 V=800.0 PL=8
MOVL C00247 V=800.0 PL=8
MOVL C00248 V=800.0 PL=8
SPYOF
MOVL C00249 V=800.0 PL=0
MOVJ C00250 VJ=25.00 PL=0
MOVL C00251 V=800.0 PL=8
SPYON
MOVL C00252 V=800.0 PL=8
MOVL C00253 V=800.0 PL=8
MOVL C00254 V=800.0 PL=8
MOVL C00255 V=800.0 PL=8
MOVL C00256 V=800.0 PL=8
MOVL C00257 V=800.0 PL=8
MOVL C00258 V=800.0 PL=8
MOVL C00259 V=800.0 PL=8
MOVL C00260 V=800.0 PL=8
MOVL C00261 V=800.0 PL=8
MOVL C00262 V=800.0 PL=8
MOVL C00263 V=800.0 PL=8
MOVL C00264 V=800.0 PL=8
MOVL C00265 V=800.0 PL=8
MOVL C00266 V=800.0 PL=8
MOVL C00267 V=800.0 PL=8
MOVL C00268 V=800.0 PL=8
MOVL C00269 V=800.0 PL=8
MOVL C00270 V=800.0 PL=8
MOVL C00271 V=800.0 PL=8
MOVL C00272 V=800.0 PL=8
MOVL C00273 V=800.0 PL=8
MOVL C00274 V=800.0 PL=8
MOVL C00275 V=800.0 PL=8
MOVL C00276 V=800.0 PL=8
MOVL C00277 V=800.0 PL=8
MOVL C00278 V=800.0 PL=8
MOVL C00279 V=800.0 PL=8
MOVL C00280 V=800.0 PL=8
MOVL C00281 V=800.0 PL=8
MOVL C00282 V=800.0 PL=8
MOVL C00283 V=800.0 PL=8
MOVL C00284 V=800.0 PL=8
MOVL C00285 V=800.0 PL=8
MOVL C00286 V=800.0 PL=8
MOVL C00287 V=800.0 PL=8
MOVL C00288 V=800.0 PL=8
SPYOF
MOVL C00289 V=800.0 PL=0
MOVJ C00290 VJ=25.00 PL=0
MOVL C00291 V=800.0 PL=8
SPYON
MOVL C00292 V=800.0 PL=8
MOVL C00293 V=800.0 PL=8
MOVL C00294 V=800.0 PL=8
MOVL C00295 V=800.0 PL=8
MOVL C00296 V=800.0 PL=8
MOVL C00297 V=800.0 PL=8
MOVL C00298 V=800.0 PL=8
MOVL C00299 V=800.0 PL=8
MOVL C00300 V=800.0 PL=8
MOVL C00301 V=800.0 PL=8
MOVL C00302 V=800.0 PL=8
MOVL C00303 V=800.0 PL=8
MOVL C00304 V=800.0 PL=8
MOVL C00305 V=800.0 PL=8
MOVL C00306 V=800.0 PL=8
MOVL C00307 V=800.0 PL=8
MOVL C00308 V=800.0 PL=8
MOVL C00309 V=800.0 PL=8
MOVL C00310 V=800.0 PL=8
MOVL C00311 V=800.0 PL=8
MOVL C00312 V=800.0 PL=8
MOVL C00313 V=800.0 PL=8
MOVL C00314 V=800.0 PL=8
MOVL C00315 V=800.0 PL=8
MOVL C00316 V=800.0 PL=8
MOVL C00317 V=800.0 PL=8
MOVL C00318 V=800.0 PL=8
MOVL C00319 V=800.0 PL=8
MOVL C00320 V=800.0 PL=8
MOVL C00321 V=800.0 PL=8
MOVL C00322 V=800.0 PL=8
MOVL C00323 V=800.0 PL=8
MOVL C00324 V=800.0 PL=8
MOVL C00325 V=800.0 PL=8
MOVL C00326 V=800.0 PL=8
MOVL C00327 V=800.0 PL=8
MOVL C00328 V=800.0 PL=8
SPYOF
MOVL C00329 V=800.0 PL=0
MOVJ C00330 VJ=25.00 PL=0
MOVL C00331 V=800.0 PL=8
SPYON
MOVL C00332 V=800.0 PL=8
MOVL C00333 V=800.0 PL=8
MOVL C00334 V=800.0 PL=8
MOVL C00335 V=800.0 PL=8
MOVL C00336 V=800.0 PL=8
MOVL C00337 V=800.0 PL=8
MOVL C00338 V=800.0 PL=8
MOVL C00339 V=800.0 PL=8
MOVL C00340 V=800.0 PL=8
MOVL C00341 V=800.0 PL=8
MOVL C00342 V=800.0 PL=8
MOVL C00343 V=800.0 PL=8
MOVL C00344 V=800.0 PL=8
MOVL C00345 V=800.0 PL=8
MOVL C00346 V=800.0 PL=8
MOVL C00347 V=800.0 PL=8
MOVL C00348 V=800.0 PL=8
MOVL C00349 V=800.0 PL=8
MOVL C00350 V=800.0 PL=8
MOVL C00351 V=800.0 PL=8
MOVL C00352 V=800.0 PL=8
MOVL C00353 V=800.0 PL=8
MOVL C00354 V=800.0 PL=8
MOVL C00355 V=800.0 PL=8
MOVL C00356 V=800.0 PL=8
MOVL C00357 V=800.0 PL=8
MOVL C00358 V=800.0 PL=8
MOVL C00359 V=800.0 PL=8
MOVL C00360 V=800.0 PL=8
MOVL C00361 V=800.0 PL=8
MOVL C00362 V=800.0 PL=8
MOVL C00363 V=800.0 PL=8
MOVL C00364 V=800.0 PL=8
MOVL C00365 V=800.0 PL=8
MOVL C00366 V=800.0 PL=8
MOVL C00367 V=800.0 PL=8
MOVL C00368 V=800.0 PL=8
MOVL C00369 V=800.0 PL=8
SPYOF
MOVL C00370 V=800.0 PL=0
MOVJ C00371 VJ=25.00 PL=0
MOVL C00372 V=800.0 PL=8
SPYON
MOVL C00373 V=800.0 PL=8
MOVL C00374 V=800.0 PL=8
MOVL C00375 V=800.0 PL=8
MOVL C00376 V=800.0 PL=8
MOVL C00377 V=800.0 PL=8
MOVL C00378 V=800.0 PL=8
MOVL C00379 V=800.0 PL=8
MOVL C00380 V=800.0 PL=8
MOVL C00381 V=800.0 PL=8
MOVL C00382 V=800.0 PL=8
MOVL C00383 V=800.0 PL=8
MOVL C00384 V=800.0 PL=8
MOVL C00385 V=800.0 PL=8
MOVL C00386 V=800.0 PL=8
MOVL C00387 V=800.0 PL=8
MOVL C00388 V=800.0 PL=8
MOVL C00389 V=800.0 PL=8
MOVL C00390 V=800.0 PL=8
MOVL C00391 V=800.0 PL=8
MOVL C00392 V=800.0 PL=8
MOVL C00393 V=800.0 PL=8
MOVL C00394 V=800.0 PL=8
MOVL C00395 V=800.0 PL=8
MOVL C00396 V=800.0 PL=8
MOVL C00397 V=800.0 PL=8
MOVL C00398 V=800.0 PL=8
MOVL C00399 V=800.0 PL=8
MOVL C00400 V=800.0 PL=8
MOVL C00401 V=800.0 PL=8
MOVL C00402 V=800.0 PL=8
MOVL C00403 V=800.0 PL=8
MOVL C00404 V=800.0 PL=8
MOVL C00405 V=800.0 PL=8
MOVL C00406 V=800.0 PL=8
MOVL C00407 V=800.0 PL=8
MOVL C00408 V=800.0 PL=8
MOVL C00409 V=800.0 PL=8
MOVL C00410 V=800.0 PL=8
MOVL C00411 V=800.0 PL=8
MOVL C00412 V=800.0 PL=8
MOVL C00413 V=800.0 PL=8
SPYOF
MOVL C00414 V=800.0 PL=0
MOVJ C00415 VJ=25.00 PL=0
MOVL C00416 V=800.0 PL=8
SPYON
MOVL C00417 V=800.0 PL=8
MOVL C00418 V=800.0 PL=8
MOVL C00419 V=800.0 PL=8
MOVL C00420 V=800.0 PL=8
MOVL C00421 V=800.0 PL=8
MOVL C00422 V=800.0 PL=8
MOVL C00423 V=800.0 PL=8
MOVL C00424 V=800.0 PL=8
MOVL C00425 V=800.0 PL=8
MOVL C00426 V=800.0 PL=8
MOVL C00427 V=800.0 PL=8
MOVL C00428 V=800.0 PL=8
MOVL C00429 V=800.0 PL=8
MOVL C00430 V=800.0 PL=8
MOVL C00431 V=800.0 PL=8
MOVL C00432 V=800.0 PL=8
MOVL C00433 V=800.0 PL=8
MOVL C00434 V=800.0 PL=8
MOVL C00435 V=800.0 PL=8
MOVL C00436 V=800.0 PL=8
MOVL C00437 V=800.0 PL=8
MOVL C00438 V=800.0 PL=8
MOVL C00439 V=800.0 PL=8
MOVL C00440 V=800.0 PL=8
MOVL C00441 V=800.0 PL=8
MOVL C00442 V=800.0 PL=8
MOVL C00443 V=800.0 PL=8
MOVL C00444 V=800.0 PL=8
MOVL C00445 V=800.0 PL=8
MOVL C00446 V=800.0 PL=8
MOVL C00447 V=800.0 PL=8
MOVL C00448 V=800.0 PL=8
MOVL C00449 V=800.0 PL=8
MOVL C00450 V=800.0 PL=8
MOVL C00451 V=800.0 PL=8
MOVL C00452 V=800.0 PL=8
MOVL C00453 V=800.0 PL=8
MOVL C00454 V=800.0 PL=8
MOVL C00455 V=800.0 PL=8
MOVL C00456 V=800.0 PL=8
MOVL C00457 V=800.0 PL=8
SPYOF
MOVL C00458 V=800.0 PL=0
MOVJ C00459 VJ=25.00 PL=0
MOVL C00460 V=800.0 PL=8
SPYON
MOVL C00461 V=800.0 PL=8
MOVL C00462 V=800.0 PL=8
MOVL C00463 V=800.0 PL=8
MOVL C00464 V=800.0 PL=8
MOVL C00465 V=800.0 PL=8
MOVL C00466 V=800.0 PL=8
MOVL C00467 V=800.0 PL=8
MOVL C00468 V=800.0 PL=8
MOVL C00469 V=800.0 PL=8
MOVL C00470 V=800.0 PL=8
MOVL C00471 V=800.0 PL=8
MOVL C00472 V=800.0 PL=8
MOVL C00473 V=800.0 PL=8
MOVL C00474 V=800.0 PL=8
MOVL C00475 V=800.0 PL=8
MOVL C00476 V=800.0 PL=8
MOVL C00477 V=800.0 PL=8
MOVL C00478 V=800.0 PL=8
MOVL C00479 V=800.0 PL=8
MOVL C00480 V=800.0 PL=8
MOVL C00481 V=800.0 PL=8
MOVL C00482 V=800.0 PL=8
MOVL C00483 V=800.0 PL=8
MOVL C00484 V=800.0 PL=8
MOVL C00485 V=800.0 PL=8
MOVL C00486 V=800.0 PL=8
MOVL C00487 V=800.0 PL=8
MOVL C00488 V=800.0 PL=8
MOVL C00489 V=800.0 PL=8
MOVL C00490 V=800.0 PL=8
MOVL C00491 V=800.0 PL=8
MOVL C00492 V=800.0 PL=8
MOVL C00493 V=800.0 PL=8
MOVL C00494 V=800.0 PL=8
MOVL C00495 V=800.0 PL=8
MOVL C00496 V=800.0 PL=8
SPYOF
MOVL C00497 V=800.0 PL=0
MOVJ C00498 VJ=25.00 PL=0
MOVL C00499 V=800.0 PL=8
SPYON
MOVL C00500 V=800.0 PL=8
MOVL C00501 V=800.0 PL=8
MOVL C00502 V=800.0 PL=8
MOVL C00503 V=800.0 PL=8
MOVL C00504 V=800.0 PL=8
MOVL C00505 V=800.0 PL=8
MOVL C00506 V=800.0 PL=8
MOVL C00507 V=800.0 PL=8
MOVL C00508 V=800.0 PL=8
MOVL C00509 V=800.0 PL=8
MOVL C00510 V=800.0 PL=8
SPYOF
MOVL C00511 V=800.0 PL=0
MOVJ C00512 VJ=25.00 PL=0
MOVL C00513 V=800.0 PL=8
SPYON
MOVL C00514 V=800.0 PL=8
MOVL C00515 V=800.0 PL=8
MOVL C00516 V=800.0 PL=8
MOVL C00517 V=800.0 PL=8
MOVL C00518 V=800.0 PL=8
SPYOF
MOVL C00519 V=800.0 PL=0
MOVJ C00520 VJ=25.00 PL=0
MOVL C00521 V=800.0 PL=8
SPYON
MOVL C00522 V=800.0 PL=8
MOVL C00523 V=800.0 PL=8
MOVL C00524 V=800.0 PL=8
MOVL C00525 V=800.0 PL=8
MOVL C00526 V=800.0 PL=8
SPYOF
MOVL C00527 V=800.0 PL=0
MOVJ C00528 VJ=25.00 PL=0
MOVL C00529 V=800.0 PL=8
SPYON
MOVL C00530 V=800.0 PL=8
MOVL C00531 V=800.0 PL=8
MOVL C00532 V=800.0 PL=8
MOVL C00533 V=800.0 PL=8
MOVL C00534 V=800.0 PL=8
SPYOF
MOVL C00535 V=800.0 PL=0
MOVJ C00536 VJ=25.00 PL=0
'Path End
MOVJ C00537 VJ=100.00 PL=0
END
